FUNCTION_BLOCK T_AddPackModeSetsCorrectly EXTENDS T_UnitTestBase
VAR
  mockState : T_MockStateModule;
  modeManager : T_ModeManager(mockState);

  maintenanceMode : T_BaseMode;
  productionMode : T_BaseMode;
  manualMode : T_BaseMode;

  actualMaintenanceMode, actualProdMode, actualManualMode : I_PackMode;
  expectedMaintenanceMode, expectedProdMode, expectedManualMode : I_PackMode;

  maintenanceResult, productionResult, manualResult : BOOL;
END_VAR

//act
modemanager.AddPackModes(productionMode, maintenanceMode, manualMode);

actualMaintenanceMode := modeManager.MaintenanceMode;
actualProdMode := modeManager.ProductionMode;
actualManualMode := modeManager.ManualMode;
expectedMaintenanceMode := maintenanceMode;
expectedProdMode := productionMode;
expectedManualMode := manualMode;

maintenanceResult := actualMaintenanceMode = expectedMaintenanceMode;
productionResult := actualProdMode = expectedProdMode;
manualResult := actualManualMode = expectedManualMode;

//asert
assertion.AssertEquals_BOOL(TRUE, maintenanceResult, 'maintenanceResult := modeManager.MaintenanceMode = maintenanceMode');
assertion.AssertEquals_BOOL(TRUE, productionResult, 'productionResult := modeManager.ProductionMode = productionMode');
assertion.AssertEquals_BOOL(TRUE, manualResult, 'manualResult := modeManager.ManualMode = manualMode');
TestFinished();

END_FUNCTION_BLOCK

(* stored: Version 1.1.0.1, ProductVersion 3.1.4024.12
   POU T_AddPackModeSetsCorrectly: Id {b4da4a75-bd92-4e63-be2c-5d78a1decb96}, SpecialFunc None *)
